Staubli VAL3: TrajSmallBox.pjx

--- TrajSmallBox.pjx ---
Parameters version=s7.6.3 stackSize=5000 millimeterUnit=true
Data file=TrajSmallBox.dtx

--- TrajSmallBox.dtx ---
mdesc mNomSpeed
public num nIndexGun
public num nKeySafeNum[6]
public num nTolKeySafeNum[6]
  [0] = 50
  [1] = 50
  [2] = 50
  [3] = 50
  [4] = 50
  [5] = 50
public num nToSafePtType
public num nToSafeFrmZ
public bool bMountOnWall
public num nRe_Tool_Z_Dits = 100
public bool bReverse_Tool_Z
public num nRe_Tool_Z_WrdZ
public num nToSafeFrmX
public num nToSafeFrmY
public num nRe_Tool_Z_WrdX
public num nRe_Tool_Z_WrdY
public pointRx pToSafePt = {fatherId=world[0]}
public jointRx jToHome
public bool bMoveJHomeJoint = true
public pointRx pPointRx = {fatherId=world[0]}
public string comment
public num nToolType
